TYPE ST_ProductRobotRecipe :
STRUCT
	wsCaption											:	WSTRING;	//	Nazwa stacji	
	                                                                      	
	stPickOffsetX									:	ST_LrParametr;	//	Offset poz pobierania x 1mm
	stPickOffsetY									:	ST_LrParametr;	//	Offset poz pobierania x 1mm
	stPickOffsetZ									:	ST_LrParametr;	//	Offset poz pobierania x 1mm
	stPickOffsetA									:	ST_LrParametr;	//	Offset poz pobierania x 1 stopeń
	stPickOffsetB									:	ST_LrParametr;	//	Offset poz pobierania x 1 stopeń
	stPickOffsetC									:	ST_LrParametr;	//	Offset poz pobierania x 1 stopeń
	                                                                      	
	stPickAccelecation								:	ST_UdiParametr;	//	Acc in % [1..100]
	stPickDecceleration								:	ST_UdiParametr;	//	Dec in % [1..100]
	stPickOverride									:	ST_UdiParametr;	//	Override in % [1..100]
	stPickColisionDetect							:	ST_UdiParametr; //	Col awoid in %[1..100]
	stPickGripperDelayTime							:	ST_UdiParametr;	//	Czas dojazdu   ms
	stSuckingTimeOn									:	ST_UdiParametr;	//	Czas posysania ms
	stSuckingTimeOff								:	ST_UdiParametr; //	Czas posysania ms
                                                                          	
	stPlaceOffsetX									:	ST_LrParametr;	//	Offset poz odkladania 2 x 1mm
	stPlaceOffsetY									:	ST_LrParametr;	//	Offset poz odkladania 2 x 1mm
	stPlaceOffsetZ									:	ST_LrParametr;	//	Offset poz odkladania 2 x 1mm
	stPlaceOffsetA									:	ST_LrParametr;	//	Offset poz odkladania 2 x 1 stopeń
	stPlaceOffsetB									:	ST_LrParametr;	//	Offset poz odkladania 2 x 1 stopeń
	stPlaceOffsetC									:	ST_LrParametr;	//	Offset poz odkladania 2 x 1 stopeń
                                                                          	
	stPlaceAccelecation								:	ST_UdiParametr;	//	Acc in % [1..100]
	stPlaceDecceleration							:	ST_UdiParametr;	//	Dec in % [1..100]
	stPlaceOverride									:	ST_UdiParametr;	//	Override in % [1..100]
	stPlaceColisionDetect							:	ST_UdiParametr; //	Col awoid in %[1..100]
	stRezerwa1										:	ST_UdiParametr;	//	
	stRezerwa2										:	ST_UdiParametr; //	
	stRezerwa3										:	ST_UdiParametr;	//	
	                                                                      	
	stDistanceTCP_X									:	ST_LrParametr; 	//	Parameter TCP narżędzia mm
	stDistanceTCP_Y									:	ST_LrParametr; 	//	Parameter TCP narżędzia mm
	stDistanceTCP_Z									:	ST_LrParametr; 	//	Parameter TCP narżędzia mm
	
	stPickPreX										:	ST_LrParametr;	//	Odsuniecie przed pozycją pobierania w osi X      
	stPickPreY										:	ST_LrParametr;	//	Odsuniecie przed pozycją pobierania w osi Y      	
	stPickPreZ										:	ST_LrParametr;	//	Odsuniecie przed pozycją pobierania w osi Z      
	stPickAfterX									:	ST_LrParametr;  //	Odsuniecie po pobraniu w osi X                   
	stPickAfterY		                            :	ST_LrParametr;  //	Odsuniecie po pobraniu w osi Y                   
	stPickAfterZ		                            :	ST_LrParametr;  //	Odsuniecie po pobraniu w osi Z                   
	stAfterPickSafeX								:	ST_LrParametr;	//	Pozycja zezwolenia wjazdu kolejenego rządu
	stPlacePreX										:	ST_LrParametr;  //	Odsuniecie przed pozycją odłożenia w osi X       
	stPlacePreY		                                :	ST_LrParametr;  //	Odsuniecie przed pozycją odłożenia w osi Y       
	stPlacePreZ		                                :	ST_LrParametr;  //	Odsuniecie przed pozycją odłożenia w osi Z       
	stPlaceAfterX		                            :	ST_LrParametr;  //	Odsuniecie po odłożenia w osi X                  
	stPlaceAfterY		                            :	ST_LrParametr;  //	Odsuniecie po odłożenia w osi Y                  
	stPlaceAfterZ		                            :	ST_LrParametr;  //	Odsuniecie po odłożenia w osi Z                  
	stProductHighOffsetZ	                        :	ST_LrParametr;  //	Wysokość produktu do ominięcia dla powrotu       
	stProductPickHeight								:	ST_LrParametr; 
END_STRUCT
END_TYPE

(* stored: Version 1.1.0.1, ProductVersion 3.1.4026.13, FileIdentifier 714f45634a5d8d06eb2671856f33dbc52d2537b2, FileSignature a476b2447aef19f20a9f8cceb0c36514757572f0154025cf8853156b4884b6ab5eb97c724b834c7d1bcf05389da88a0d4258ab36aea0f135545ada78e859278c1699676e9446d997ecf4f129184c14cc3526848c1c504372f88b470321435856534118e33262b299aa77ab8834e7c5ed3bb1309e4c0d6a1ff77681df621d0e5c4621e3110d7aaec003d63ec2df901827821f0abe0dcfa72d62dd7187f4e26e23f0f9114aaa0ed421ec3fe8f32d173163885e9e544f20cb64a1af88e0e40f9807aee1504d639af086731aeb6a037930c4eba5ae680818c4430ebd62dc2eb753465ede1b9ed7f3533ab220c767ed1752dc3ac620cf3036f12c4714de3ea52b4fc7
   DUT ST_ProductRobotRecipe: Id {86acee25-814f-4fa6-aca4-6fcf89afc5fc} *)
